Staubli VAL3: addStrArray1.pgx

public program addStrArray1(string& x_sStrIn[], num x_nPos, num x_nNum, bool& x_bRes)
  local num l_i
begin
  //建立指定数目的字符串数组
  //x_sStrIn:返回的新数组
  //x_nPos：指定位置
  //x_nNum:数组个数
  //x_bRes:函数返回值
  x_bRes=false
  if x_nNum<1
    popUpMsg("新增点个数小于1")
    return
  endIf
  if x_nPos<0
    x_nPos=0
  else
    if x_nPos>size(x_sStrIn)
      x_nPos=size(x_sStrIn)
    endIf
  endIf
  //取整
  x_nNum=roundDown(x_nNum)
   //插入新数据
  for l_i=x_nPos+1 to x_nPos+x_nNum
    insert(x_sStrIn[l_i])
  endFor
  x_bRes=true
end
